TYPE T_Ctrl_SIf_STB_In :
STRUCT
	/// Sensor hanger detected
	bolHangerDetected: T_Ctrl_IoBoolDebounced;
	/// Sensor buffer full
	bolBufferFull: T_Ctrl_IoBoolDebounced;
	/// Sensor decrement counter (option)
	bolDecrementCounter: T_Ctrl_IoBoolDebounced;
END_STRUCT
END_TYPE

(* stored: Version 1.1.0.1, ProductVersion 3.1.0.23
   DUT T_Ctrl_SIf_STB_In: Id {d0ec1f95-4508-48eb-9394-02595bb2b07d} *)
